Omron CX-Programmer project NewProject (CX-Programmer 9.75)

# PLC NewPLC1: CP1H XA

## Global symbols (name address type ; comment)
0.02 BOOL  ; Latch
0.03 BOOL  ; Unlatch
0.07 BOOL  ; ENABLE
0.08 BOOL  ; SW1
0.09 BOOL  ; SW2
100.04 BOOL  ; Motor
Motor_ONOFF Automation_process
QIS Automation_process
QIS2 Automation2
QIS3 IF_ELSIF

## Program NewProgram1 (cyclic task 0)
Local symbols
DO1 D1 UINT
DO2 D2 UINT
DO5 D5 UINT
DO6 D6 UINT

### Section Section1

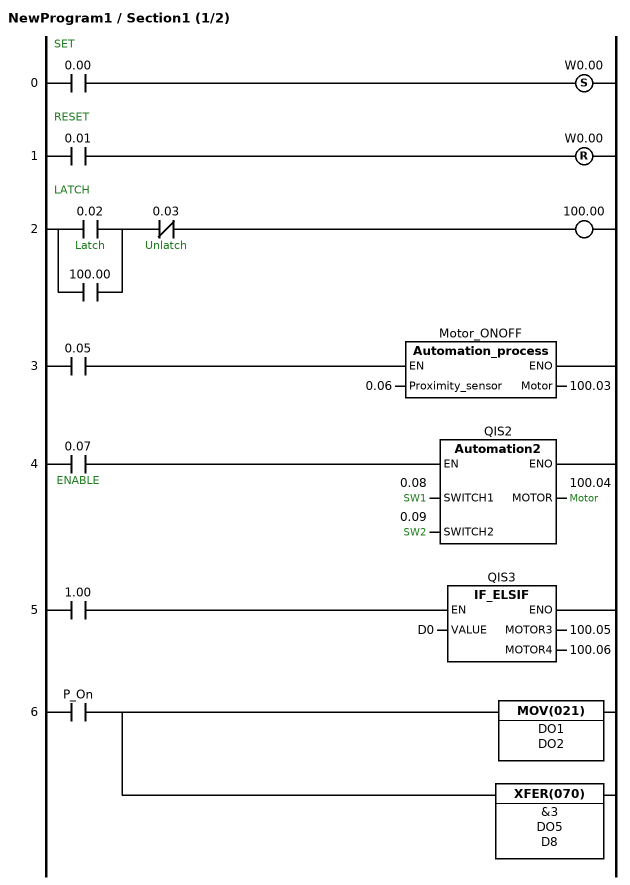
; rung 0: SET
LD 0.00
SET W0.00
; rung 1: RESET
LD 0.01
RSET W0.00
; rung 2: LATCH
LD 0.02  ; Latch
OR 100.00
ANDNOT 0.03  ; Unlatch
OUT 100.00
; rung 3
LD 0.05
CALL Motor_ONOFF : Automation_process (Proximity_sensor := 0.06, Motor => 100.03)
; rung 4
LD 0.07  ; ENABLE
CALL QIS2 : Automation2 (SWITCH1 := 0.08, SWITCH2 := 0.09, MOTOR => 100.04)  ; SW1, SW2, Motor
; rung 5
LD 1.00
CALL QIS3 : IF_ELSIF (VALUE := D0, MOTOR3 => 100.05, MOTOR4 => 100.06)
; rung 6
LD P_On
MOV(021) DO1 DO2
XFER(070) &3 DO5 D8

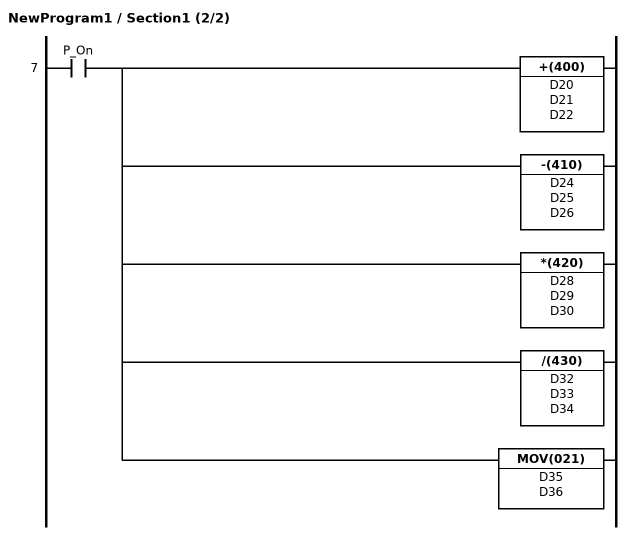
; rung 7
LD P_On
+(400) D20 D21 D22
-(410) D24 D25 D26
*(420) D28 D29 D30
/(430) D32 D33 D34
MOV(021) D35 D36

### Section END
; rung 0
END(001)

## Function block Automation2
VAR_INPUT
  SWITCH1 : BOOL;
  SWITCH2 : BOOL;
END_VAR
VAR_OUTPUT
  MOTOR : BOOL;
END_VAR
IF SWITCH1 = TRUE THEN
	MOTOR := TRUE;
END_IF;
IF SWITCH2 = TRUE THEN
	MOTOR := FALSE;
END_IF;

## Function block Automation_process
VAR_INPUT
  Proximity_sensor : BOOL;
END_VAR
VAR_OUTPUT
  Motor : BOOL;
END_VAR
IF Proximity_sensor = TRUE  THEN
	Motor := TRUE;
	
ELSE
	Motor := FALSE;
END_IF;

## Function block IF_ELSIF
VAR_INPUT
  VALUE : UINT;
END_VAR
VAR_OUTPUT
  MOTOR3 : BOOL;
  MOTOR4 : BOOL;
END_VAR
IF VALUE = 1 THEN
	MOTOR3 := TRUE;
	MOTOR4 := FALSE;
ELSIF VALUE = 2 THEN
	MOTOR3 := FALSE;
	MOTOR4 := TRUE;
ELSE
	MOTOR3 := FALSE;
	MOTOR4 := FALSE;
END_IF;